FUNCTION_BLOCK TcoQlSetCommandTask EXTENDS TcoQlSeriesSupplyTask
VAR
    _command : TcoQlSeriesSupply_SetControl_v_1_x_x;
END_VAR

SUPER^(inoConfig := inoConfig, inoStatus := inoStatus);

(*~
    <docu>
        <summary>
            Restores this instance to the Ready state. Can be called explicitly or from within one of the restore mechanisms.
            <para>
                See also <see cref="PlcDocu.TcoCore.TcoTask.AutoRestorable()"/>
            </para>
        </summary>
    </docu>
~*)
METHOD Restore : ITcoRestorable
SUPER^.Restore();
END_METHOD

METHOD WithParams : REFERENCE TO TcoQlSetCommandTask
VAR_INPUT
    inCommand : TcoQlSeriesSupply_SetControl_v_1_x_x;
END_VAR
THIS^._command := inCommand;
WithParams REF= THIS^;
END_METHOD

END_FUNCTION_BLOCK

(* stored: Version 1.1.0.1, ProductVersion 3.1.4024.12
   POU TcoQlSetCommandTask: Id {d98c79d9-a8e3-0ee9-2151-213862bbf5d2}, SpecialFunc None
   Method Restore: Id {0057f43e-d449-071b-33fe-e154bdf4f389}
   Method WithParams: Id {ca3b81ee-b772-00dd-13b7-6d078aa4bf4a} *)
